FUNCTION WithinTolerance : BOOL
VAR_INPUT
	value : LREAL;
	target : LREAL;
	tolerance : LREAL;
END_VAR
(*
checks if value is close enough to target within a given margin
*)

WithinTolerance := ABS(value-target) < tolerance;

END_FUNCTION

(* stored: Version 1.1.0.1, ProductVersion 3.1.4024.11
   POU WithinTolerance: Id {70d5a386-b333-45cf-9af1-a80becc50e58}, SpecialFunc None *)
